FUNCTION TryConvert_USINT_TO_BOOL : BOOL
VAR_INPUT
	in : USINT;
	out : REFERENCE TO BOOL;
END_VAR

out := USINT_TO_BOOL(in);
TryConvert_USINT_TO_BOOL := TRUE;

END_FUNCTION

(* stored: Version 1.1.0.1, ProductVersion 3.1.4024.12
   POU TryConvert_USINT_TO_BOOL: Id {a03889f5-a9b4-42ac-b789-76e2a70626ae}, SpecialFunc None *)
